// TIA Portal V17 export
// export: Created 2025-08-05T09:35:59.9677351Z, ExportSetting WithDefaults, DisplayName Totally Integrated Automation Portal, DisplayVersion V17, DisplayName TIA Portal Openness, DisplayVersion V17, DisplayName TIA Portal Version Control Interface, DisplayVersion V17, DisplayName SINAMICS Startdrive Advanced, DisplayVersion V17, DisplayName SINAMICS Startdrive G130, G150, S120, S150, SINAMICS MV, S210, DisplayVersion V17, DisplayName SINAMICS Startdrive G110M, G120, G120C, G120D, G120P, G115D, DisplayVersion V17, DisplayName STEP 7 Professional, DisplayVersion V17, DisplayName STEP 7 Safety, DisplayVersion V17, DisplayName WinCC Advanced, DisplayVersion V17
TYPE "typeGroupOvrvListEntry"
TITLE = Entry group overview / Eintrag Gruppenübersicht
// Entry group overview [V 01.00 | Kernel_V2] / Eintrag Gruppenübersicht [V 01.00 | Kernel_V2]
// stored: IsFailsafeCompliant false
   STRUCT
      alive : USInt;   // Alive-Flag (Wird in der Gruppe gesetzt, zentral dann zurückgesetzt) / Alive-Flag (is set in group, then centrally reset)
      dbAnyAddr : DB_ANY;   // DB-Any Adresse (typeCaCgFg) / DB any address (typeCaCgFg)
      nextPartnerIndex : DInt := -1;   // Index der Nächsten Partner-Gruppe / Index of next partner group
      firstChildIndex : DInt := -1;   // Index der ersten untergeordneten Gruppe / Index of first subordinate group
   END_STRUCT;
END_TYPE
